(* CoDeSys 2.3.9.62 project: Semaforos.pro *)
(* Libraries: Util.lib*26.9.14 10:12:46, Standard.lib 4.10.05 10:14:46, IecSfc.lib*2.6.14 10:37:46 *)

(* Global variable list: Global_Variables *)
VAR_GLOBAL

    (* Entradas *)
     Interr:BOOL;
     Normal:BOOL;

     (* Salidas *)
     S1RV:BOOL;              (* Semaforo 1 Rojo  Vehículos*)
     S1AV:BOOL;              (*  Semaforo 1 Ambar Vehículos*)
     S1VV:BOOL;               (* Semaforo 1 Verde Vehículos*)
     S1RP: BOOL;            (* Semaforo 1 Rojo Peatones*)
     S1VP:BOOL;           (* Semaforo 1 Verde Peatones*)

    S2RV:BOOL;              (* Semaforo 2 Rojo  Vehículos*)
     S2AV:BOOL;              (*  Semaforo 2 Ambar Vehículos*)
     S2VV:BOOL;               (* Semaforo 2 Verde Vehículos*)
    S2RP: BOOL;        (* Semaforo 2 Rojo Peatones*)
     S2VP:BOOL;          (* Semaforo 2 Verde Peatones*)

END_VAR

(* POU PLC_PRG, ST *)
PROGRAM PLC_PRG
VAR

END_VAR

END_PROGRAM

(* POU Intermitente, LD *)
FUNCTION_BLOCK Intermitente
VAR_INPUT
	Habilita:BOOL;
	Tiempo_alto:TIME;
	Tiempo_bajo:TIME;

END_VAR
VAR_OUTPUT
	Salida:BOOL;

END_VAR
VAR
	E0: BOOL;
	Eon: BOOL;
	tempAlto: TON;
	Eoff: BOOL;
	tempBajo: TON;
END_VAR
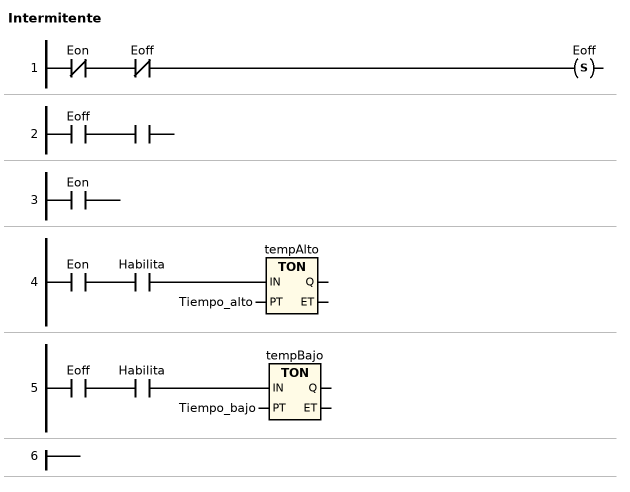
_LD_ (* Ladder Diagram *)
NETWORK 1
	[/Eon] - [/Eoff] --- (S Eoff)
NETWORK 2
	[Eoff] - []
NETWORK 3
	[Eon]
NETWORK 4
	[Eon] - [Habilita] - tempAlto:TON(IN: *, PT: Tiempo_alto)
NETWORK 5
	[Eoff] - [Habilita] - tempBajo:TON(IN: *, PT: Tiempo_bajo)
NETWORK 6
	*
_END_LD_
(* the same logic as Structured Text *)
(* Network 1 *)
IF NOT Eon AND NOT Eoff THEN Eoff := TRUE; END_IF;
(* Network 2: see the listing above *)
(* Network 3: see the listing above *)
(* Network 4 *)
tempAlto(IN := Eon AND Habilita, PT := Tiempo_alto);
(* Network 5 *)
tempBajo(IN := Eoff AND Habilita, PT := Tiempo_bajo);
(* Network 6: see the listing above *)
END_FUNCTION_BLOCK

(* Visualisation Cruce
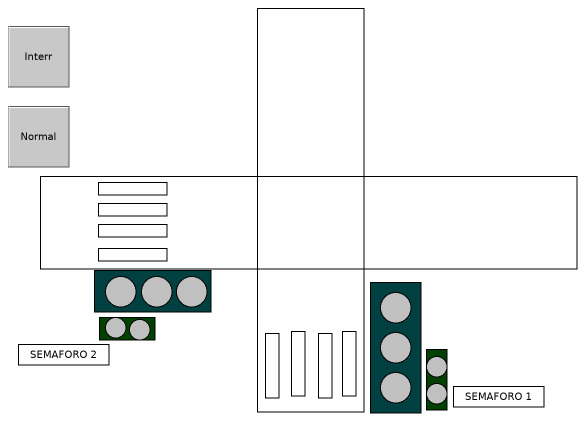
button at (20,50)-(81,111): text "Interr"; toggles Interr
button at (20,130)-(81,191): text "Normal"; toggles Normal
ellipse at (392,316)-(423,347): alarm colour if S1RV
ellipse at (392,356)-(423,387): alarm colour if S1AV
ellipse at (392,396)-(423,427): alarm colour if S1VV
ellipse at (438,380)-(459,401): alarm colour if S1RP
ellipse at (438,407)-(459,428): alarm colour if S1VP
ellipse at (188,300)-(219,331): alarm colour if S2RV
ellipse at (153,300)-(184,331): alarm colour if S2AV
ellipse at (117,300)-(148,331): alarm colour if S2VV
ellipse at (141,343)-(162,364): alarm colour if S2RP
ellipse at (117,341)-(138,362): alarm colour if S2VP
rectangle at (465,410)-(556,431): text "SEMAFORO 1"
rectangle at (30,368)-(121,389): text "SEMAFORO 2"
14 more shapes without text or variables
*)

(* Visualisation Semaforo
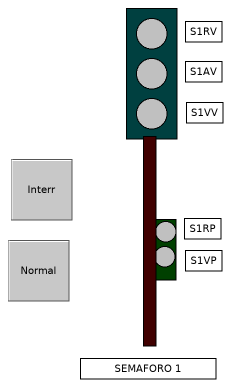
button at (38,186)-(99,247): text "Interr"; toggles Interr
button at (35,267)-(96,328): text "Normal"; toggles Normal
ellipse at (163,45)-(194,76): alarm colour if S1RV
ellipse at (163,85)-(194,116): alarm colour if S1AV
ellipse at (163,125)-(194,156): alarm colour if S1VV
ellipse at (182,248)-(203,269): alarm colour if S1RP
ellipse at (181,273)-(202,294): alarm colour if S1VP
rectangle at (212,48)-(249,69): text "S1RV"
rectangle at (212,88)-(249,109): text "S1AV"
rectangle at (213,129)-(250,150): text "S1VV"
rectangle at (211,245)-(248,266): text "S1RP"
rectangle at (212,277)-(249,298): text "S1VP"
rectangle at (107,385)-(243,406): text "SEMAFORO 1"
3 more shapes without text or variables
*)
